Fanuc KAREL source: kb00066.KL

-- PROVISIONAL review KL for V940-1; original PC SHA256 01164074b6c0730abbc45fd37b79a6bb9ca4aac408ba15ac7f6c29c37afab839
-- Incomplete behavior may be omitted. Consult companion uncertainty JSON. Do not deploy.
PROGRAM KB00066
%NOLOCKGROUP
BEGIN
  -- V9_ZERO_TABLE_METADATA_HINT layout=0002_ascii; no indexed target words; source/name/runtime held
  -- UNRESOLVED_PC offsets 5-14; opcodes 3F,75
  -- UNRESOLVED_PC offsets 19-26; opcodes 9D,23
  -- UNRESOLVED_PC offsets 31-38; opcodes 9D,23
  -- UNRESOLVED_PC offsets 43-50; opcodes 9D,23
  -- UNRESOLVED_PC offsets 55-62; opcodes 9D,23
  -- UNRESOLVED_PC offsets 67-74; opcodes 9D,23
  -- UNRESOLVED_PC offsets 79-139; opcodes 27,22,2A,22,22,22,22,22,22,22,22,31
  -- UNRESOLVED_PC offsets 144-148; opcodes 7F
END KB00066
